(* IEC 61131-3 sources: OpenPLC61850/webserver/st_files, 3 files *)

(* ---- 209569.st ---- *)
PROGRAM boiler
  VAR
    raw_pressure AT %IW100 : INT := 3100;
    setpoint AT %QW1 : INT := 3000;
    efflux AT %QX0.0 : BOOL;
  END_VAR
  VAR
    _TMP_GT1_OUT : BOOL;
  END_VAR

  _TMP_GT1_OUT := GT(raw_pressure, setpoint);
  efflux := _TMP_GT1_OUT;
END_PROGRAM

CONFIGURATION Config0

  RESOURCE Res0 ON PLC
    TASK task0(INTERVAL := T#20ms,PRIORITY := 0);
    PROGRAM instance0 WITH task0 : boiler;
  END_RESOURCE
END_CONFIGURATION

(* ---- 853040.st ---- *)
PROGRAM boiler
  VAR
    raw_pressure AT %QW2 : INT := 3100;
    setpoint AT %QW1 : INT := 3000;
    efflux AT %QX0.0 : BOOL;
  END_VAR
  VAR
    _TMP_GT1_OUT : BOOL;
  END_VAR

  _TMP_GT1_OUT := GT(raw_pressure, setpoint);
  efflux := _TMP_GT1_OUT;
END_PROGRAM

CONFIGURATION Config0

  RESOURCE Res0 ON PLC
    TASK task0(INTERVAL := T#20ms,PRIORITY := 0);
    PROGRAM instance0 WITH task0 : boiler;
  END_RESOURCE
END_CONFIGURATION

(* ---- blank_program.st ---- *)
PROGRAM prog0
  VAR
    var_in : BOOL;
    var_out : BOOL;
  END_VAR

  var_out := var_in;
END_PROGRAM

CONFIGURATION Config0

  RESOURCE Res0 ON PLC
    TASK Main(INTERVAL := T#50ms,PRIORITY := 0);
    PROGRAM Inst0 WITH Main : prog0;
  END_RESOURCE
END_CONFIGURATION
